// TwinCAT 3 PLC project Punzonatrice_2223
// ProgramVersion: 3.1.4024.0
// libraries:
//   Tc2_Standard, * (Beckhoff Automation GmbH)
//   Tc2_System, * (Beckhoff Automation GmbH)
//   Tc3_Module, * (Beckhoff Automation GmbH)
// project tree:
//   GVLs/ GVL_HMI.TcGVL, GVL_IO.TcGVL
//   / PlcTask.TcTTO
//   POUs/ FB_MSF.TcPOU, FB_oscillatore.TcPOU, MAIN.TcPOU
// real-time tasks:
//   TASK PlcTask: cycle T#10ms, priority 20, ADS port 350

CONFIGURATION Punzonatrice_2223
    RESOURCE PLC ON TwinCAT3
        TASK PlcTask(INTERVAL := T#10ms, PRIORITY := 20);
        PROGRAM MAIN WITH PlcTask : MAIN;
    END_RESOURCE
END_CONFIGURATION

// ---- GVLs/GVL_HMI.TcGVL
{attribute 'qualified_only'}
// GVL_HMI
VAR_GLOBAL
	// ingressi da HMI
	hmi_start: BOOL;
	hmi_stop: BOOL := TRUE;
	hmi_ack: BOOL;
	
	// uscite verso HMI
	hmi_lstart: BOOL;
	hmi_lstop: BOOL;
	hmi_lack: BOOL;
	msg_stato:	STRING(21) :='';
END_VAR

// ---- GVLs/GVL_IO.TcGVL
{attribute 'qualified_only'}
// GVL_IO
VAR_GLOBAL
	// pulsante start - I5
	PSTART	AT %I*:BOOL;
	// pulsante stop (NC) - I6
	PSTOP	AT %I*:BOOL;
	// pulsante ripristino - I7
	PACK	AT %I*:BOOL;
	// pulsante emergenza (NC) - I8
	PEMERG	AT %I*:BOOL;
	// Sensore ingresso nastro (NC) - I1
	I1		AT %I*:BOOL;
	// Sensore pezzo in posizione (NC) - I2
	I2		AT %I*:BOOL;
	// Sensore mandrino in alto - I3
	I3		AT %I*:BOOL;
	// Sensore mandrino in basso - I4
	I4		AT %I*:BOOL;
	// Motore avanzamento nastro, caricamento pezzo - Q1
	Q1		AT %Q*:BOOL;
	// Motore ritorno nastro, scarico pezzo - Q2
	Q2		AT %Q*:BOOL;
	// Motore salita mandrino - Q3
	Q3		AT %Q*:BOOL;
	// Motore discesa mandrino - Q4
	Q4		AT %Q*:BOOL;
	// Indicatore start - Q5
	LSTART	AT %Q*:BOOL;
	// Indicatore stop - Q6
	LSTOP	AT %Q*:BOOL;
	// Indicatore ack - Q7
	LACK	AT %Q*:BOOL;	
END_VAR

// ---- POUs/MAIN.TcPOU
PROGRAM MAIN
VAR
	punzonatrice	:	FB_MSF();
END_VAR

//eseguo l'istanza della punzonatrice
punzonatrice(
	start:= GVL_IO.PSTART, 
	stop:= GVL_IO.PSTOP, 
	ack:= GVL_IO.PACK, 
	emerg:= GVL_IO.PEMERG, 
	i1:= GVL_IO.I1, 
	i2:= GVL_IO.I2, 
	i3:= GVL_IO.I3, 
	i4:= GVL_IO.I4, 
	q1=> GVL_IO.Q1, 
	q2=> GVL_IO.Q2, 
	q3=> GVL_IO.Q3, 
	q4=> GVL_IO.Q4, 
	lstart=> GVL_IO.LSTART, 
	lstop=> GVL_IO.LSTOP, 
	lack=> GVL_IO.LACK);

END_PROGRAM

// ---- POUs/FB_MSF.TcPOU
FUNCTION_BLOCK FB_MSF
VAR_INPUT
	start	:	BOOL;
	stop	:	BOOL;
	ack		:	BOOL;
	emerg	:	BOOL;
	i1		:	BOOL;
	i2		:	BOOL;
	i3		:	BOOL;
	i4		:	BOOL;
END_VAR
VAR_OUTPUT
	q1		:	BOOL;
	q2		:	BOOL;
	q3		:	BOOL;
	q4		:	BOOL;
	lstart	:	BOOL;
	lstop	:	BOOL;
	lack	:	BOOL;
END_VAR
VAR
	// enumeratore privato degli stati, la variabile stato parte da S0
	stato : (S0, S1, S2, S3, S4, S5, S6, S7, S8, SE, SA) := S0;
	//timer T34 attesa dopo caricamento
	T34		:	TON();
	T82		:	TON();
	
	//bit di abilitazione
	enable	:	BOOL;
	
	//bit delle transizioni
	tr_01	:	BOOL;
	tr_02	:	BOOL;
	tr_12	:	BOOL;
	tr_23	:	BOOL;
	tr_34	:	BOOL;
	tr_45	:	BOOL;
	tr_56	:	BOOL;
	tr_67	:	BOOL;
	tr_78	:	BOOL;
	tr_80	:	BOOL;
	tr_82	:	BOOL;
	tr_EA	:	BOOL;
	tr_A0	:	BOOL;
	
	//memoria dello stop nominale
	mArresto	:	BOOL := FALSE;
	
	//memoria di un pezzo in lavorazione sul nastro
	mPezzoCarico	:	BOOL := FALSE;
	
	// lampeggio
	osc : FB_oscillatore();
END_VAR

// 1. aggiornamento condizioni di abilitazione
enable := stop AND emerg;

// 2. aggiornamento timers, contatori, triggers sui fronti
T34(IN := (stato = S3 AND enable), PT := T#2S );
T82(IN := (stato = S8 AND enable), PT := T#3S );
osc(enable := (stato=SA) OR (stato = SE), t_high := T#500MS, t_low := T#500MS);

// 3. valutazione della condizione di arresto nominale
IF NOT stop AND emerg THEN
	IF (stato = S1 OR stato = S2) THEN
		stato := S0;
	ELSIF (stato = S3 OR stato = S4 OR stato = S5 OR stato = S6 OR stato = S7 OR stato = S8) THEN
		mArresto := TRUE;
	END_IF
END_IF

// 4. valutazione della condizione di arresto di emergenza
IF NOT emerg THEN
	stato := SE;
END_IF

// 5. aggiornamento delle condizioni di transizione di stato
tr_01 := enable AND NOT(i3) AND start;
tr_02 := enable AND i3 AND start;
tr_12 := enable AND i3;
tr_23 := enable AND i1;
tr_34 := enable AND T34.Q AND NOT (i1);
tr_45 := enable AND NOT (i2);
tr_56 := enable AND i4;
tr_67 := enable AND i3;
tr_78 := enable AND NOT (I1);
tr_82 := enable AND T82.Q AND NOT mArresto AND i1;
tr_80 := enable AND mArresto;

//comando uscite
lstart := (stato <> S0);
lstop := (stato = S0) OR ((stato = SE) AND osc.Q);
lack := (stato = SE) OR ((stato = SA) AND osc.Q);
q1 := (stato = S4);
q2 := (stato = S7) OR ((stato = SA) AND mPezzoCarico);
q3 := (stato = S1) OR (stato = S6) OR ((stato = SA) AND NOT (i3));
q4 := (stato = S5);

END_FUNCTION_BLOCK

// ---- POUs/FB_oscillatore.TcPOU
FUNCTION_BLOCK FB_oscillatore
VAR_INPUT
	enable	: BOOL;
	t_high	: TIME;
	t_low	: TIME;	
END_VAR
VAR_OUTPUT
	q		: BOOL;	
END_VAR
VAR
	t1		: TON();
	t2		: TON();	
END_VAR

t1(in := enable AND NOT t2.Q, pt := t_low);
t2(in := t1.Q, pt := t_high);
// comando dell'uscita dell'oscillatore
q := t1.Q;

END_FUNCTION_BLOCK
